// TIA Portal V20 export
VAR_GLOBAL   // PLC tag table "IO_PLC_Functinal_Test_1_PLC_Functinal_Test_3"
   In_Functional_Test AT %I300.0 : "IO_Device_Functinal_Test";
   Out_Test_Parameters AT %Q300.0 : "IO_Device_Test_Parameters";
END_VAR
